PROGRAM MAIN
VAR
END_VAR

END_PROGRAM

(* stored: Version 1.1.0.1
   POU MAIN: Id {9cd90b6c-bf45-4cd8-a7f2-47ed1148f8a8}, SpecialFunc None *)
